# B&R Automation Studio project Parker_BMM_ST_V5_3147_V12 (part 19)

#### scrshot.c
```c
/********************************************************************
 * COPYRIGHT --  B&R China
 ********************************************************************
 * Program: length
 * File: length.c
 * Author: lijianjun
 * Created: March 06, 2013
 ********************************************************************
 * Implementation of program length --- parison length control
 ********************************************************************/

#include <bur/plctypes.h>

#ifdef _DEFAULT_INCLUDES
	#include <AsDefault.h>
#endif

#include <string.h>

/* Description: 	screen shot	(C language)	Library - VCScrsht										           */
/*------------------------------------------------------------------------------------------------------*/
/*				这个任务必须在循环7任务里，而且循环7的循环周期必须是1000ms，冗余时间为1000ms			       */
/*				It must also be inserted into Task Class #7 [1000 ms] and have a tolerance of 1000 ms.      */
/*  			程序员需要在初始化任务里定义device名称及相关信息就好了									           */
/*------------------------------------------------------------------------------------------------------*/
/*	version		author			date			decription
*********************************************************************************************************/

/********************************************************************************************************/
/*	<|> Variable to control this task:																                    */
/*		Name							Typ					Description									                    */
/*		step							| UINT				| screen shot step							                 //
//		DateTimeString_0			| DateTimeString	| output current date and time as string	              //
//		more see variable declaration																	                    */
/********************************************************************************************************/

/********************************************************************************************************/
/*	State commentary:																					      //
//			INIT:					   init step															   //
//			WAIT_USB_INSERT:		wait usb device insert												//
//			WAIT_COMMAND:    		wait for command													   //
//			INIT_SCREEN_SHOT:		Init screen shot													   //
//			SCREEN_SHOT:			Screen shot															   //
//			DEINIT_SCREEN_SHOT:		DeInit																//
//			ERROR_STEP:				Error step															   */

/********************************************************************************************************/
/*  Others:
//		指定首选存储介质:																				         //
//          在CPU属性里My Device定义介质名称															    //

//		截屏产生的文件名格式，以当前日期时间为文件名的bmp文件，DateTimeString_0.Date_Mode:		//
//				1:		美国时间格式USA date format  -- DateMM-DD-YYYY_TimeHH-MM-SS					  //
//				2:		亚洲时间格式Asia date format -- DateYYYY-MM-DD_TimeHH-MM-SS					  //
//				others:	默认模式Default format       -- DateDD-MM-YYYY_TimeHH-MM-SS				 //

//		建议：用fileio库来判断所在介质中是否有相同名称的文件，防止被覆盖								//
//		suggest: use filio to judge whether have a same name files in current diretory		  //

//		截屏状态gScreenShot.Status																		       //
//			0		等待存储介质插入插槽
			1		等待截屏开始指令
			2		截屏中
			3		截屏出错																			             //

*********************************************************************************************************/

/**********************************************************************************
**                          函数声明											 **
**********************************************************************************/

/**********************************************************************************
**                          宏定义												 **
**********************************************************************************/
#define INIT				         		0
#define WAIT_USB_INSERT		      		10
#define WAIT_DIR_SCREEN_CREATE		   20
#define WAIT_DIR_SINGLE_CREATE			40
#define WAIT_DIR_ALL_CREATE	   		50

#define WAIT_COMMAND		         100
#define INIT_SCREEN_SHOT	      110
#define SCREEN_SHOT			      120
#define DEINIT_SCREEN_SHOT	      140
#define ERROR_STEP			      200

/**********************************************************************************
**     	        		任务初始化								 				 **
**********************************************************************************/

_INIT  	void init()
{
	/*--------- 程序员根据实际，需要修改的代码 开始 ---------*/

	strcpy(gUSB_1.DeviceName, "USB_1");		/* 指定首选存储介质 */
	strcpy(gUSB_2.DeviceName, "USB_2");		/* 指定第二个选择存储介质 */

   strcpy(gUSB_1.DirScreenDeviceName, "SCREEN_1");		/* 指定首选存储介质目录 */
   strcpy(gUSB_2.DirScreenDeviceName, "SCREEN_2");		/* 指定第二个选择存储介质目录 */

   strcpy(dirScreenName,"ScreenShot");
   strcpy(dirSingleName,"SingleRecipe");
   strcpy(dirAllName,"AllRecipe");

   strcpy(gUSB_1.DirSingleDeviceName, "SINGLE_1");		/* 指定首选存储介质目录 */
   strcpy(gUSB_2.DirSingleDeviceName, "SINGLE_2");		/* 指定第二个选择存储介质目录 */

   strcpy(gUSB_1.DirAllDeviceName, "ALL_1");		/* 指定首选存储介质目录 */
   strcpy(gUSB_2.DirAllDeviceName, "ALL_2");		/* 指定第二个选择存储介质目录 */

	DateTimeString_0.Date_Mode = 2;		 	/* 截屏产生的文件名格式，见上面的说明 */

	statusUSB1 = 0;
	statusUSB2 = 0;

	gUSB_1.reserve = 0;
	gUSB_2.reserve = 0;

	/*--------- 程序员根据实际，需要修改的代码 结束 ---------*/
}/* _INIT  	void init() */

/**********************************************************************************
**     	        		任务循环部分							 				 **
**********************************************************************************/
_CYCLIC void cyclic()
{
   STRING NumName[5];

	/* 接收截屏开始指令 在别的任务里定义，原因：这个任务周期太长，有时抓不到信号 */
	gScreenShot.CmdScreenShot = gScreenShot.CmdScreenShot;

	gScreenShot.Status = gScreenShot.Status;/* 对外接口，截屏状态 */

	/*judge have a usb device insert or not*/
	/* 判断存储介质是否插入插槽内 */
	DirInfo_1.enable= 1;
	DirInfo_1.pDevice= (UDINT)(&gUSB_1.DeviceName);	/* 首选存储介质 */
	DirInfo_1.pPath= 0;							/* For Root, pPath is 0 */

	DirInfo(&DirInfo_1);

	if(DirInfo_1.status != ERR_FUB_BUSY)
	{
		if(DirInfo_1.status == ERR_OK)
		{
			statusUSB1 = 1;
		}
		else
		{
			if(DirInfo_1.status == fiERR_SYSTEM && ERR_FUB_BUSY == FileIoGetSysError())
			{
				statusUSB1 = 1;
			}
			else
			{
				statusUSB1 = 0;  /*  no usb  */
				gUSB_1.DeviceOk = 0;
				gUSB_1.reserve = 0;
			}
		}
	}/* if(DirInfo_1.status != ERR_FUB_BUSY) */

	if(1 == statusUSB1 && 0 == statusUSB1_old)
	{
		gUSB_1.reserve = 1;
	}

	statusUSB1_old = statusUSB1;

	DirInfo_2.enable= 1;
	DirInfo_2.pDevice= (UDINT)(&gUSB_2.DeviceName);
	DirInfo_2.pPath= 0;

	DirInfo(&DirInfo_2);

	if(DirInfo_2.status != ERR_FUB_BUSY)
	{
		if(DirInfo_2.status == ERR_OK)
		{
			statusUSB2 = 1;
		}
		else
		{
			if(DirInfo_2.status == fiERR_SYSTEM && ERR_FUB_BUSY == FileIoGetSysError())
			{
				statusUSB2 = 1;
			}
			else
			{
				statusUSB2 = 0;   /*  no usb  */
				gUSB_2.DeviceOk = 0;
				gUSB_2.reserve = 0;
			}
		}
	}/* if(DirInfo_2.status != ERR_FUB_BUSY) */

	if(1 == statusUSB2 && 0 == statusUSB2_old)
	{
		gUSB_2.reserve = 1;
	}

   if(0 == gUSB_2.DeviceOk && 0 == gUSB_1.DeviceOk)
   {
      if(1 == gScreenShot.CmdScreenShot)
      {
         gImply.NoUSB = 1;
         gScreenShot.CmdScreenShot = 0;
      }
   }
	/* 不在等待截屏指令状态， 如果谁发了截屏指令，无效 */
	if(gScreenShot.Status != 1)
	{
		gScreenShot.CmdScreenShot = 0;
		HideButton =1; //ipis1226
	}
	else
	{
		HideButton =0;	//ipis1226
	}

	/* 所有设备都没有准备好，就停在等待存储介质插入步 */
	if((gUSB_1.reserve == 0) && (gUSB_2.reserve == 0))
	{
		step = WAIT_USB_INSERT;
	}

	switch(step)
	{
		case INIT:				/* Init */
			gScreenShot.Status = 0;	/* 等待存储介质插入插槽 */
			step = WAIT_USB_INSERT;
			break;

		case WAIT_USB_INSERT:	/* wait for usb device insert */
			gScreenShot.Status = 0;	/* 等待存储介质插入插槽 */

			step = step;

			if((gUSB_1.reserve == 1) || (gUSB_2.reserve == 1))
			{
				step = WAIT_DIR_SCREEN_CREATE;
			}
			break;

      case WAIT_DIR_SCREEN_CREATE:
         if(gUSB_1.reserve == 1)
         {
            strcpy(deviceName, gUSB_1.DeviceName);
         }
         else if(gUSB_2.reserve == 1)
         {
            strcpy(deviceName, gUSB_2.DeviceName);
         }
         DirCreate_1.enable = 1;
         DirCreate_1.pDevice= (UDINT)(&deviceName);
         DirCreate_1.pName  = (UDINT)(&dirScreenName);

         /* Call FBK */
         DirCreate(&DirCreate_1);

         if(ERR_OK == DirCreate_1.status || fiERR_DIR_ALREADY_EXIST == DirCreate_1.status)
         {
            DirCreate_1.enable = 0;
            step = WAIT_DIR_SINGLE_CREATE;
         }
         else if(DirCreate_1.status != ERR_FUB_BUSY)
         {
				if(0 == strcmp(deviceName, gUSB_1.DeviceName))gUSB_1.reserve = 0;
				if(0 == strcmp(deviceName, gUSB_2.DeviceName))gUSB_2.reserve = 0;

            DirCreate_1.enable = 0;
            step = INIT;
         }
         break;

      case WAIT_DIR_SINGLE_CREATE:
         if(gUSB_1.reserve == 1)
         {
            strcpy(deviceName, gUSB_1.DeviceName);
         }
         else if(gUSB_2.reserve == 1)
         {
            strcpy(deviceName, gUSB_2.DeviceName);
         }
         DirCreate_1.enable = 1;
         DirCreate_1.pDevice= (UDINT)(&deviceName);
         DirCreate_1.pName  = (UDINT)(&dirSingleName);

         /* Call FBK */
         DirCreate(&DirCreate_1);

         if(ERR_OK == DirCreate_1.status || fiERR_DIR_ALREADY_EXIST == DirCreate_1.status)
         {
            DirCreate_1.enable = 0;
            step = WAIT_DIR_ALL_CREATE;
         }
         else if(DirCreate_1.status != ERR_FUB_BUSY)
         {
				if(0 == strcmp(deviceName, gUSB_1.DeviceName))gUSB_1.reserve = 0;
				if(0 == strcmp(deviceName, gUSB_2.DeviceName))gUSB_2.reserve = 0;

            DirCreate_1.enable = 0;
            step = INIT;
         }
         break;

      case WAIT_DIR_ALL_CREATE:
         if(gUSB_1.reserve == 1)
         {
            strcpy(deviceName, gUSB_1.DeviceName);
         }
         else if(gUSB_2.reserve == 1)
         {
            strcpy(deviceName, gUSB_2.DeviceName);
         }
         DirCreate_1.enable = 1;
         DirCreate_1.pDevice= (UDINT)(&deviceName);
         DirCreate_1.pName  = (UDINT)(&dirAllName);

         /* Call FBK */
         DirCreate(&DirCreate_1);

         if(ERR_OK == DirCreate_1.status || fiERR_DIR_ALREADY_EXIST == DirCreate_1.status)
         {
				if(0 == strcmp(deviceName, gUSB_1.DeviceName))gUSB_1.DeviceOk = 1;
				if(0 == strcmp(deviceName, gUSB_2.DeviceName))gUSB_2.DeviceOk = 1;

            DirCreate_1.enable = 0;
            step = WAIT_COMMAND;
         }
         else if(DirCreate_1.status != ERR_FUB_BUSY)
         {
				if(0 == strcmp(deviceName, gUSB_1.DeviceName))gUSB_1.reserve = 0;
				if(0 == strcmp(deviceName, gUSB_2.DeviceName))gUSB_2.reserve = 0;

            DirCreate_1.enable = 0;
            step = INIT;
         }
         break;

		case WAIT_COMMAND:		/* Wait for command */

			gScreenShot.Status = 1;	/* 等待截屏开始指令 */

			/* 允许客户按截屏开始按键 */
			gScreenShot.ScreenShotBtnStatus = gScreenShot.ScreenShotBtnStatus & (65535-2);

			if(gScreenShot.CmdScreenShot == 1)
			{
				gScreenShot.CmdScreenShot = 0;

				gScreenShot.ScreenShotBtnStatus = gScreenShot.ScreenShotBtnStatus | 2;

				/* Name format of Screen file: Year-month-day-hour-minute-second.bmp */
				DateTimeString_0.enable = 1;
				/*DateTimeString_0.Date_Mode = 2;		 Asia mode: DateYYYY-MM-DD_TimeHH-MM-SS */

            itoa((long)(gPanelObj.GetPicture),(unsigned long)NumName);

            strcpy(scrshotFileName,"Page_");

            strcat(scrshotFileName,NumName);

            strcat(scrshotFileName, "_");

            DateTimeString(&DateTimeString_0);

            strcat(scrshotFileName, DateTimeString_0.DisplayString);

            strcat(scrshotFileName, ".bmp");

				if(gUSB_1.DeviceOk == 1)
				{
					strcpy(deviceName, gUSB_1.DirScreenDeviceName);
				}
				else if(gUSB_2.DeviceOk == 1)
				{
					strcpy(deviceName, gUSB_2.DirScreenDeviceName);
				}
				step = INIT_SCREEN_SHOT;
			}
			break;

		case INIT_SCREEN_SHOT:	/* Init screen shot */

			gScreenShot.Status = 2;	/* 截屏中 */

			status = InitScreenShot(1, (UDINT)(&pHandle), (UDINT)(&scrshotFileName), (UDINT)(&deviceName), (UDINT)(&gPanelObj.VisualName));
			if(status == 0)
			{
				step = SCREEN_SHOT;
			}
			else
			{
				gScreenShot.errorNumber = status;
				step = ERROR_STEP;
			}
			break;

		case SCREEN_SHOT:		/* Screen shot */

			status = ScreenShot(1, pHandle);

			if(status != 1001)
			{
				if(status == 0)
				{
					step = DEINIT_SCREEN_SHOT;
				}
				else
				{
					gScreenShot.errorNumber = status;
					step = ERROR_STEP;
				}
			}
			break;

		case DEINIT_SCREEN_SHOT:/* DeInit screen shot */

			status = DeInitScreenShot(1, pHandle);

			if(status == 0)
			{
				step = WAIT_COMMAND;
			}
			else
			{
				gScreenShot.errorNumber = status;
				step = ERROR_STEP;
			}
			break;

		case ERROR_STEP:		/* Error step */

			gScreenShot.Status = 3;	/* 截屏出错 */
			step = INIT;
			break;
	}/* switch(step) */
}/* _CYCLIC void cyclic() */
```

#### scrshot.var
```iecst
VAR
	step : UINT;
	statusUSB1 : USINT;
	statusUSB1_old : USINT;
	statusUSB2 : USINT;
	statusUSB2_old : USINT;
	scrshotFileName : STRING[59];
	deviceName : STRING[19];
	DateTimeString_0 : DateTimeString;
	pHandle : UDINT;
	DirInfo_1 : DirInfo;
	DirInfo_2 : DirInfo;
	DirCreate_1 : DirCreate;
	dirScreenName : STRING[19];
	dirSingleName : STRING[19];
	dirAllName : STRING[19];
	status : UINT;
	HideButton : USINT; (*ipis1226*)
END_VAR
```

### Program Logical/screen/password (ANSIC, version 1.00.0) - password login modify

#### password.c
```c
/********************************************************************
 * COPYRIGHT --  B&R China
 ********************************************************************
 * Program: password
 * File: password.c
 * Author: lijianjun
 * Created: March 06, 2013
 ********************************************************************
 * Implementation of program password --- password control
 ********************************************************************/

#include <bur/plctypes.h>
#include <string.h>

#ifdef _DEFAULT_INCLUDES
	#include <AsDefault.h>
#endif

#include "pic_id.h"

/**************************************************************************************
** 					 	 dedine								              			 **
**************************************************************************************/
#define S$STEP_INIT_OK     10000

#define S$STEP_IDLE        100
#define S$STEP_READ        1000
#define S$STEP_WRITE       2000

#define S$STEP_ERROR	      30000

/**************************************************************************************
** 							         function declare  				  			             **
**************************************************************************************/
void Pwd_Set(unsigned short picGet,unsigned short  picObj);
/**************************************************************************************
*     	        		      I N I T U P  O F   T H E   T A S K 		 				       **
**************************************************************************************/

_INIT  void Pwd_init( void )
{
	InputCompletion = 0;

	strcpy(gPwd.PwdInput,   "           ");    	/*  11 space char  */
	strcpy(gPwd.HisPwdInput,"           ");		/*  11 space char  */

	DataObjOperate.InitStep = 100;
}
/**************************************************************************************
*        				    C Y C L I C   P A R T   O F   T H E   T A S K  				  *
**************************************************************************************/

_CYCLIC  void Pwd_cyclic ( void )
{

	if (gPasswordLogout)  //ipis0218
	{
		InputCompletion =1;
		strcpy(gPwd.PwdInput,   "           ");    	/*  11 space char  */
		gPasswordLogout =0;
	}

	gPanelObj.PasswordLevel = gPwd.PwdLevel;

	switch(DataObjOperate.InitStep)
	{
		case 100:
			DataObjOperate.Ident = 0;

			DatObj_Info.enable = 1;
			DatObj_Info.pName  =(unsigned long)("pwddata");
			DatObjInfo(&DatObj_Info);

			if(doERR_MODULNOTFOUND == DatObj_Info.status)
			{
				DataObjOperate.InitStep = 200;
			}
			else if(0 == DatObj_Info.status)
			{
				DataObjOperate.Ident    = DatObj_Info.ident;
				DataObjOperate.InitStep = 800;
			}
			else
			{
				DataObjOperate.InitStep = S$STEP_ERROR;
			}
			break;
		case 200:                              	/* create data module */
			DatObj_Create.enable   = 1;
			DatObj_Create.pName    = DatObj_Info.pName;
			DatObj_Create.len      = sizeof(Pwd_typ);
			DatObj_Create.MemType  = doUSRROM;
			DatObj_Create.Option   = 0;
			DatObj_Create.pCpyData = 0;

			DataObjOperate.InitStep = 300;
			break;
		case 300:
			DatObjCreate(&DatObj_Create);
			if(0 == DatObj_Create.status)
			{
				DataObjOperate.Ident = DatObj_Create.ident;
				DataObjOperate.InitStep = 400;
			}
			break;
		case 400:
			memset(&gPwd,0,sizeof(Pwd_typ));

			strcpy(gPwd.Level[2],"8888");
			strcpy(gPwd.Level[1],"7777");
			strcpy(gPwd.Level[0],"6666");

			gPwd.length_1 = 120;
			gPwd.length_2 = 120;
			gPwd.length_3 = 120;

			strcpy(gPwd.Pwd_1,"0098768876");
			strcpy(gPwd.Pwd_2,"0098768872");
			strcpy(gPwd.Pwd_3,"0098768870");

			strcpy(gPwd.PwdInput,   "           ");    	 	 /*  11 space char  */
			strcpy(gPwd.HisPwdInput,"           ");			/*  11 space char  */

			DataObjOperate.InitStep = 500;
			break;
		case 500:
			DatObj_Write.enable  = 1;
			DatObj_Write.ident	 = DataObjOperate.Ident;
			DatObj_Write.pSource = (unsigned long )&gPwd;
			DatObj_Write.len     = sizeof(Pwd_typ);

			DataObjOperate.InitStep = 600;
			break;
		case 600:
			DatObjWrite(&DatObj_Write);
			if(0 == DatObj_Write.status)
			{
				DataObjOperate.InitStep = 700;
			}
			else
			{
				DataObjOperate.InitStep = S$STEP_ERROR;
			}
			break;
		case 700:
			DataObjOperate.InitStep = 1000;
			break;
		case 800:
			DatObj_Read.enable 		 = 1;
			DatObj_Read.ident 		 = DataObjOperate.Ident ;
			DatObj_Read.Offset 		 = 0;
			DatObj_Read.pDestination = (unsigned long )&gPwd;
			DatObj_Read.len 		 = sizeof(Pwd_typ);

			DataObjOperate.InitStep = 900;
			break;
		case 900:
			DatObjRead(&DatObj_Read);
			if(0 == DatObj_Read.status)
			{
				DataObjOperate.InitStep = 1000;
			}
			else
			{
				DataObjOperate.InitStep = S$STEP_ERROR;
			}
			break;
		case 1000:
			gPwd.PwdLevel = 0;

			strcpy(gPwd.PwdInput,   "           ");    	/*  11 space char  */
			strcpy(gPwd.HisPwdInput,"           ");	    /*  11 space char  */

			DataObjOperate.Step = S$STEP_IDLE;
			DataObjOperate.InitStep = S$STEP_INIT_OK;
			break;
		case S$STEP_ERROR:
			break;
		default:
			break;
	}/* switch(DataObjOperate.InitStep) */

	if(DataObjOperate.Ident != 0 && DataObjOperate.InitStep == S$STEP_INIT_OK )
	{
		switch(DataObjOperate.Step )
		{
			case S$STEP_IDLE:
				if(1 == gPwd.wSavePassword)
				{
					gPwd.wSavePassword = 0;
					DataObjOperate.Step = S$STEP_WRITE;
				}
				break;
			case S$STEP_WRITE:
				DatObj_Write.enable  = 1;
				DatObj_Write.ident	 = DataObjOperate.Ident;
				DatObj_Write.pSource = (unsigned long )&gPwd;
				DatObj_Write.len     = sizeof(Pwd_typ);

				DataObjOperate.Step = S$STEP_WRITE + 100;
				break;
			case (S$STEP_WRITE + 100):
				DatObjWrite(&DatObj_Write);
				if(0 == DatObj_Write.status)
				{
					DataObjOperate.Step = S$STEP_WRITE + 200;
				}
				break;
			case (S$STEP_WRITE + 200):
				DataObjOperate.Step = S$STEP_IDLE;
				break;
			default:
				break;
		}/* switch(DataObjOperate.Step) */

		WorkingDays = 0;

		if(1 == gPwd.Option[0] && 0 == gPwd.OK_1)
		{
			WorkingDays = WorkingDays + gPwd.length_1;
		}
		else if(1 == gPwd.Option[1] && 0 == gPwd.OK_2)
		{
			WorkingDays = WorkingDays + gPwd.length_2;
		}
		else if(1 == gPwd.Option[2] && 0 == gPwd.OK_3)
		{
			WorkingDays = WorkingDays + gPwd.length_3;
		}

		if(0 == WorkingDays)
		{
			gMachineInfo.TimeStopMachine = 0;
		}
		else
		{
			if(gMachineStopDays > WorkingDays)
			{
				gMachineInfo.TimeStopMachine = 1;
			}
			else
			{
				gMachineInfo.TimeStopMachine = 0;
			}
		}

		if(gAlarm.batteryLow)
		{
			gMachineInfo.TimeStopMachine = 0;
		}

		if(PIC_PASSWORD_LOGIN == gPanelObj.GetPicture || PIC_INIT == gPanelObj.GetPicture)
		{
			if(1 == InputCompletion)
			{
				InputCompletion = 0;
				strcpy(gPwd.HisPwdInput,gPwd.PwdInput);
				strcpy(gPwd.PwdInput,"           ");		/*  11 space char  */

				if( !strcmp(gPwd.HisPwdInput,gPanelObj.PasswordHigh))
				{
			   		gPwd.PwdLevel = 5;
			   	}
				else if( !strcmp(gPwd.HisPwdInput,gPanelObj.Password4))
				{
			   		gPwd.PwdLevel = 4;
			   	}
				else if(!strcmp(gPwd.HisPwdInput,gPwd.Level[2]))
				{
					gPwd.PwdLevel = 3;
				//	gPwd.PwdLevel = 4;  //ipis0226
				}
				else if(!strcmp(gPwd.HisPwdInput,gPwd.Level[1]))
				{
					gPwd.PwdLevel = 2;
				}
				else if(!strcmp(gPwd.HisPwdInput,gPwd.Level[0]))
				{
					gPwd.PwdLevel = 1;
				}
				else
				{
					if(PIC_PASSWORD_LOGIN == gPanelObj.GetPicture)
					{
						if(!strcmp(gPwd.HisPwdInput,gPwd.Pwd_3))
						{
							if(1 == gPwd.Option[2])
							{
								gMachineStopDays = 0;
								gPwd.OK_3 = 1;
								gPwd.OK_2 = 1;
								gPwd.OK_1 = 1;
								gPwd.wSavePassword = 1;
							}
						}
						else if (!strcmp(gPwd.HisPwdInput,gPwd.Pwd_2))
						{
							if(1 == gPwd.Option[1])
							{
								gMachineStopDays = 0;
								gPwd.OK_2 = 1;
								gPwd.OK_1 = 1;
								gPwd.wSavePassword = 1;
							}
						}
						else if (!strcmp(gPwd.HisPwdInput,gPwd.Pwd_1))
						{
							if(1 == gPwd.Option[0])
							{
								gMachineStopDays = 0;
								gPwd.OK_1 = 1;
								gPwd.wSavePassword = 1;
							}
						}
					}/* if(PIC_PASSWORD_LOGIN == gPanelObj.GetPicture) */
					gPwd.PwdLevel = 0;
				}
			}/* if(1 == InputCompletion */
		}/* if(gPanelObj.GetPicture == PIC_PASSWORD_LOGIN || PIC_INIT_PIC == gPanelObj.GetPicture ) */

		Pwd_Set(gPanelObj.GetPicture,PIC_PASSWORD_SET);

	}/* if(DataObjOperate.Ident != 0 && DataObjOperate.InitStep == S$STEP_INIT_OK ) */
}
/**************************************************************************************
** 							Function Realization  				  			         **
**************************************************************************************/

void Pwd_Set(UINT picGet,UINT picObj)
{
	short	i;

 	if (picGet != picObj)
 	{
		gPwd.StatusOfPasswordSet = 0;
		for (i=0;i<=2;i++)
		{
			strcpy(gPwd.PasswordSet[i],   "           ");
			strcpy(gPwd.HisPasswordSet[i],"           ");
		}
 		return;
 	}

 	for (i=0;i<=2;i++)
 	{

 		if(1 == gPwd.CompletionHisPasswordSet[i])
 		{
 			gPwd.StatusOfPasswordSet         = 1;
 			gPwd.CompletionHisPasswordSet[i] = 0;
 		}

 		if(1 == gPwd.CompletionPasswordSet[i])
	 	{
	 		if (strcmp(gPwd.PasswordSet[i] ,"           ")!= 0)
		    {
			    if (0 == strcmp(gPwd.PasswordSet[i],gPwd.HisPasswordSet[i]))
				{
					gPwd.StatusOfPasswordSet  = 2; /* setting ok */
		    		gPwd.wSavePassword	  	 = 1;
		    		strcpy(gPwd.Level[i],gPwd.PasswordSet[i]);

					strcpy(gPwd.PasswordSet[i],   "           ");
					strcpy(gPwd.HisPasswordSet[i],"           ");

		    	}
	    		else
	    		{
	    			gPwd.StatusOfPasswordSet = 3; /* setting failed */

	 				strcpy(gPwd.PasswordSet[i],   "           ");
					strcpy(gPwd.HisPasswordSet[i],"           ");
	    		}
	    	}
			gPwd.CompletionPasswordSet[i] = 0;
	 	}/* if(1 == gPwd.CompletionPasswordSet[i]) */
	}/* for (i=0;i<=2;i++) */
 }/* end of function */
```

#### password.var
```iecst
VAR
	DatObj_Info	:DatObjInfo;
	DatObj_Create	:DatObjCreate;
	DatObj_Write	:DatObjWrite;
	DatObj_Read	:DatObjRead;
	DataObjOperate	:DatObj_Operate_typ;
    InputCompletion	:USINT;

    WorkingDays : UDINT;
END_VAR
```

### Program Logical/screen/vpn (ANSIC, version 1.00.0) - IP configure

#### vpn.c
```c
/********************************************************************
 * COPYRIGHT --  B&R China
 ********************************************************************
 * Program: vpn
 * File: vpn.c
 * Author: lijianjun
 * Created: March 06, 2013
 ********************************************************************
 * Implementation of program vpn --- ip address control
 ********************************************************************/

#include <bur/plctypes.h>

#ifdef _DEFAULT_INCLUDES
#include <AsDefault.h>
#endif

#include <string.h>

//#include "keyap880.h"
#include "keyap2100.h"
#include "pic_id.h"

char substring(char *dst,char *src,int start,int len);

/********************************************************************************************************/
/*  Others:
	vpn.FlagManualSetIP：0=自动获取IP地址类型，1=手动设置IP地址
	vpn存放当前IP地址，子网掩码，网关地址等，以及手动设置IP地址，子网掩码，网关地址等参数，

		typedef struct
		{
			BOOL			FlagManualSetIP;		* 标志位：1 = 手动设定IP地址 *
			BOOL			CmdSetIP;				* 设置IP地址指令 *
			BOOL			CmdSetSubnetMark;		* 设置子网掩码指令 *
			BOOL			CmdSetGateway;			* 设置网关地址指令 *

			STRING			CurrentIPString[16];	* 当前IP地址 *
			STRING			CurrentSubnetMarkString[16];* 当前子网掩码 *
			STRING			CurrentGatewayString[16];* 当前网关地址 *

			Address_typ		ParaSetIP;				* 手动设置IP地址模式下，IP地址参数 *
			Address_typ		ParaSetSubnetMark;		* 手动设置IP地址模式下，子网掩码参数 *
			Address_typ		ParaSetGateway;			* 手动设置IP地址模式下，网关地址参数 *

		}VPN_typ;

*********************************************************************************************************/

/**********************************************************************************
**                          宏定义												 **
**********************************************************************************/
#define INIT				       0
#define GET_ETH_CFG_MODE	   10
#define GET_ETH_CFG_ADR	      20
#define GET_ETH_CFG_SUBNET	   30
#define GET_ETH_CFG_GATEWAY 	40

#define WAIT_COMMAND          100
#define SET_ETH_CFG_MODE		110
#define SET_ETH_CFG_ADR	      120
#define SET_ETH_CFG_SUBNET 	130
#define SET_ETH_CFG_GATEWAY   140
#define ERROR_STEP            9999

/**********************************************************************************
**     	        		I N I T U P  O F   T H E   T A S K 		 				 **
**********************************************************************************/
_INIT void init()
{
	/*------------- 编程人员根据实际需要修改的地方 开始 -----------------*/

	strcpy(vpnDevice,"IF3");	/*指定VPN使用的端口*/

	/*------------- 编程人员根据实际需要修改的地方 结束 -----------------*/
	step = INIT;

	bGetCurrentIP_USINT = 1;

}/* _INIT void init() */

/**********************************************************************************
**        			C Y C L I C   P A R T   O F   T H E   T A S K  				 **
**********************************************************************************/
_CYCLIC void cyclic()
{
	if(gPanelObj.GetPicture == PIC_IP_CONFIG && step == WAIT_COMMAND)
	{
		F5_bHiden = 0;
	}
	else
	{
		F5_bHiden = 1;
	}

	/*-------------- 判断手自动模式是否切换了 -------------------------*/
	R_TRIG_KeyF5.CLK = gPanelObj.KeyMatric[S$KEYMATRIX_F5];
		R_TRIG(&R_TRIG_KeyF5);

	/*if(1 == R_TRIG_KeyF5.Q)
	{
		if(gPanelObj.GetPicture == PIC_IP_CONFIG)
		{
			if(0 == F5_bHiden)
			{
				if( cfgCONFIGMODE_MANUALLY == vpn.CurrentConfigMode)
				{
					vpn.ParaSetConfigMode = cfgCONFIGMODE_DHCPCLIENT;
				}
				else
				{
					vpn.ParaSetConfigMode = cfgCONFIGMODE_MANUALLY;
				}
				vpn.CmdSetMode = 1;
			}
		}
	}*//* if(1 == R_TRIG_KeyF5.Q) */

	vpn.ParaSetConfigMode = cfgCONFIGMODE_MANUALLY;

	switch(step)
	{
		case INIT:				/*初始化*/
			step = GET_ETH_CFG_MODE;
			break;

		case GET_ETH_CFG_MODE:	/*读当前配置模式*/
			CfgGetEthConfigMode_0.pDevice = (UDINT)&vpnDevice[0];
			CfgGetEthConfigMode_0.enable  = 1;

			CfgGetEthConfigMode(&CfgGetEthConfigMode_0);

			if(ERR_FUB_BUSY != CfgGetEthConfigMode_0.status)
			{
				if(ERR_OK == CfgGetEthConfigMode_0.status)
				{
					if(cfgCONFIGMODE_MANUALLY == CfgGetEthConfigMode_0.ConfigMode)
					{
						vpn.FlagManualSetIP = 1;
						step = GET_ETH_CFG_ADR;
					}
					else if(cfgCONFIGMODE_DHCPCLIENT == CfgGetEthConfigMode_0.ConfigMode)
					{
						vpn.FlagManualSetIP = 0;
						step = GET_ETH_CFG_ADR;
					}
					vpn.CurrentConfigMode = CfgGetEthConfigMode_0.ConfigMode;
				}
				else
				{
					step = ERROR_STEP;
				}
			}
			break;

		case GET_ETH_CFG_ADR:		/*读当前IP地址*/
			CfgGetIPAddr_0.pDevice = (UDINT)&vpnDevice[0];
			CfgGetIPAddr_0.pIPAddr = (UDINT)&vpn.CurrentIPString[0];
			CfgGetIPAddr_0.Len     = 16;
			CfgGetIPAddr_0.enable  = 1;

			CfgGetIPAddr(&CfgGetIPAddr_0);

			if(ERR_FUB_BUSY != CfgGetIPAddr_0.status)
			{
				if(ERR_OK == CfgGetIPAddr_0.status)
				{
					step = GET_ETH_CFG_SUBNET;
				}
				else
				{
					step = ERROR_STEP;
				}
			}
			break;

		case GET_ETH_CFG_SUBNET:		/*读当前子网掩码*/
			CfgGetSubnetMask_0.pDevice = (UDINT)&vpnDevice[0];
			CfgGetSubnetMask_0.pSubnetMask = (UDINT)&vpn.CurrentSubnetMarkString[0];
			CfgGetSubnetMask_0.Len     = 16;
			CfgGetSubnetMask_0.enable  = 1;

			CfgGetSubnetMask(&CfgGetSubnetMask_0);

			if(ERR_FUB_BUSY != CfgGetSubnetMask_0.status)
			{
				if(ERR_OK == CfgGetSubnetMask_0.status)
				{
					step = GET_ETH_CFG_GATEWAY;
				}
				else
				{
					step = ERROR_STEP;
				}
			}
			break;

		case GET_ETH_CFG_GATEWAY:		/*读当前默认网关*/
			CfgGetDefaultGateway_0.pDevice = (UDINT)&vpnDevice[0];
			CfgGetDefaultGateway_0.pGateway= (UDINT)&vpn.CurrentGatewayString[0];
			CfgGetDefaultGateway_0.Len     = 16;
			CfgGetDefaultGateway_0.enable  = 1;

			CfgGetDefaultGateway(&CfgGetDefaultGateway_0);

			if(ERR_FUB_BUSY != CfgGetDefaultGateway_0.status)
			{
				if(ERR_OK == CfgGetDefaultGateway_0.status)
				{
					step = WAIT_COMMAND;
				}
				else
				{
					if(cfgERR_PARAM_NOT_SET == CfgGetDefaultGateway_0.status)
					{
						step = WAIT_COMMAND;
					}
					else
					{
						step = ERROR_STEP;
					}
				}
			}
			break;

		case WAIT_COMMAND:
			if(0 == vpn.FlagManualSetIP)
			{
				vpn.CmdSetIP         = 0;
				vpn.CmdSetSubnetMark = 0;
				vpn.CmdSetGateway    = 0;

				if(1 == vpn.CmdSetMode)
				{
					vpn.CmdSetMode = 0;
					step = SET_ETH_CFG_MODE;
				}
				else
				{
					step = GET_ETH_CFG_MODE;
				}
			}
			else
			{
				if(1 == vpn.CmdSetMode)
				{
					vpn.CmdSetMode = 0;
					step = SET_ETH_CFG_MODE;
				}
				else
				{
					if(1 == vpn.CmdSetIP)
					{
						vpn.CmdSetIP = 0;
						step = SET_ETH_CFG_ADR;
					}
					else if(1 == vpn.CmdSetSubnetMark)
					{
						vpn.CmdSetSubnetMark = 0;
						step = SET_ETH_CFG_SUBNET;
					}
					else if(1 == vpn.CmdSetGateway)
					{
						vpn.CmdSetGateway = 0;
						step = SET_ETH_CFG_GATEWAY;
					}
				}/* if(1 == vpn.CmdSetMode) */
			}/* if(0 == vpn.FlagManualSetIP) */
			break;

		case SET_ETH_CFG_MODE:		/*设定配置模式*/
			CfgSetEthConfigMode_0.pDevice = (UDINT)&vpnDevice[0];

			CfgSetEthConfigMode_0.ConfigMode = vpn.ParaSetConfigMode;
			CfgSetEthConfigMode_0.Option  = cfgOPTION_VOLATILE;

			CfgSetEthConfigMode_0.enable  = 1;

			CfgSetEthConfigMode(&CfgSetEthConfigMode_0);

			if(ERR_FUB_BUSY != CfgSetEthConfigMode_0.status)
			{
				if(ERR_OK == CfgSetEthConfigMode_0.status)
				{
					step = GET_ETH_CFG_MODE;
				}
				else
				{
					step = ERROR_STEP;
				}
			}
			break;

		case SET_ETH_CFG_ADR:		/*设定IP*/
			itoa(vpn.ParaSetIP.Address3, (UDINT)&tempString);
			strcpy(setIPString, tempString);

			strcat(setIPString, ".");

			itoa(vpn.ParaSetIP.Address2, (UDINT)&tempString);
			strcat(setIPString, tempString);

			strcat(setIPString, ".");

			itoa(vpn.ParaSetIP.Address1, (UDINT)&tempString);
			strcat(setIPString, tempString);

			strcat(setIPString, ".");

			itoa(vpn.ParaSetIP.Address0, (UDINT)&tempString);
			strcat(setIPString, tempString);

			CfgSetIPAddr_0.pDevice = (UDINT)&vpnDevice[0];
			CfgSetIPAddr_0.pIPAddr = (UDINT)&setIPString[0];
			CfgSetIPAddr_0.Option  = cfgOPTION_NON_VOLATILE;
			CfgSetIPAddr_0.enable  = 1;

			CfgSetIPAddr(&CfgSetIPAddr_0);

			if(ERR_FUB_BUSY != CfgSetIPAddr_0.status)
			{
				if(ERR_OK == CfgSetIPAddr_0.status)
				{
					step = GET_ETH_CFG_MODE;

					/*update fix*/
					gUserFix.ProjectInfo.Address3 = vpn.ParaSetIP.Address3;
					gUserFix.ProjectInfo.Address2 = vpn.ParaSetIP.Address2;
					gUserFix.ProjectInfo.Address1 = vpn.ParaSetIP.Address1;
					gUserFix.ProjectInfo.Address0 = vpn.ParaSetIP.Address0;

					gRecipeOperate.OnceSave = 1;
				}
				else
				{
					step = ERROR_STEP;
				}
			}
			break;

		case SET_ETH_CFG_SUBNET:		/*设定子网掩码*/
			itoa(vpn.ParaSetSubnetMark.Address3, (UDINT)&tempString);
			strcpy(setSubnetMarkString, tempString);

			strcat(setSubnetMarkString, ".");

			itoa(vpn.ParaSetSubnetMark.Address2, (UDINT)&tempString);
			strcat(setSubnetMarkString, tempString);

			strcat(setSubnetMarkString, ".");

			itoa(vpn.ParaSetSubnetMark.Address1, (UDINT)&tempString);
			strcat(setSubnetMarkString, tempString);

			strcat(setSubnetMarkString, ".");

			itoa(vpn.ParaSetSubnetMark.Address0, (UDINT)&tempString);
			strcat(setSubnetMarkString, tempString);

			CfgSetSubnetMask_0.pDevice = (UDINT)&vpnDevice[0];
			CfgSetSubnetMask_0.pSubnetMask = (UDINT)&setSubnetMarkString[0];
			CfgSetSubnetMask_0.Option  = cfgOPTION_NON_VOLATILE;
			CfgSetSubnetMask_0.enable  = 1;

			CfgSetSubnetMask(&CfgSetSubnetMask_0);

			if(ERR_FUB_BUSY != CfgSetSubnetMask_0.status)
			{
				if(ERR_OK == CfgSetSubnetMask_0.status)
				{
					step = GET_ETH_CFG_MODE;
				}
				else
				{
					step = ERROR_STEP;
				}
			}
			break;

		case SET_ETH_CFG_GATEWAY:		/*设定网关*/
			itoa(vpn.ParaSetGateway.Address3, (UDINT)&tempString);
			strcpy(setGatewayString, tempString);

			strcat(setGatewayString, ".");

			itoa(vpn.ParaSetGateway.Address2, (UDINT)&tempString);
			strcat(setGatewayString, tempString);

			strcat(setGatewayString, ".");

			itoa(vpn.ParaSetGateway.Address1, (UDINT)&tempString);
			strcat(setGatewayString, tempString);

			strcat(setGatewayString, ".");

			itoa(vpn.ParaSetGateway.Address0, (UDINT)&tempString);
			strcat(setGatewayString, tempString);

			CfgSetDefaultGateway_0.pDevice = (UDINT)&vpnDevice[0];
			CfgSetDefaultGateway_0.pGateway = (UDINT)&setGatewayString[0];
			CfgSetDefaultGateway_0.Option  = cfgOPTION_NON_VOLATILE;
			CfgSetDefaultGateway_0.enable  = 1;

			CfgSetDefaultGateway(&CfgSetDefaultGateway_0);

			if(ERR_FUB_BUSY != CfgSetDefaultGateway_0.status)
			{
				if(ERR_OK == CfgSetDefaultGateway_0.status)
				{
					step = GET_ETH_CFG_MODE;
				}
				else
				{
					step = ERROR_STEP;
				}
			}
			break;

		case ERROR_STEP:	/*error step*/
			step = 0;
			break;

		default:
			break;
	}/* switch(step) */

	/*Get config ip*/
	if(bGetCurrentIP_USINT)
	{
		bGetCurrentIP_USINT = 0;
		Part_num_count = 0;
		Char_num = 0;
		old_Char_num = 0;
		for (ii = 0; ii < sizeof(vpn.CurrentIPString); ii++)
		{
			Charr = (char*)(vpn.CurrentIPString[ii]);

			if( Charr == 46)
			{
				Char_num = ii;

				switch (Part_num_count)
				{
					case 0:
						substring(sTempAddress3,vpn.CurrentIPString,0,Char_num);
						old_Char_num = Char_num;
						break;
					case 1:
						substring(sTempAddress2,vpn.CurrentIPString,old_Char_num+1,Char_num-old_Char_num-1);
						old_Char_num = Char_num;
						break;
					case 2:
						substring(sTempAddress1,vpn.CurrentIPString,old_Char_num+1,Char_num-old_Char_num-1);
						old_Char_num = Char_num;
						break;
				}
				Part_num_count++;
			}
			if(Part_num_count == 3)
			{
				substring(sTempAddress0,vpn.CurrentIPString,old_Char_num+1,sizeof(vpn.CurrentIPString)-old_Char_num);
			}

		}

		uConfigAddress3 = atoi((UDINT) &sTempAddress3);
		uConfigAddress2 = atoi((UDINT) &sTempAddress2);
		uConfigAddress1 = atoi((UDINT) &sTempAddress1);
		uConfigAddress0 = atoi((UDINT) &sTempAddress0);

		/*check current vs fix (if different than excute set ip cmd)*/
		if(gUserFix.ProjectInfo.Address0 != uConfigAddress0
			|| gUserFix.ProjectInfo.Address1 != uConfigAddress1
			|| gUserFix.ProjectInfo.Address2 != uConfigAddress2
			|| gUserFix.ProjectInfo.Address3 != uConfigAddress3
			)
		{
			vpn.ParaSetIP.Address0 = gUserFix.ProjectInfo.Address0;
			vpn.ParaSetIP.Address1 = gUserFix.ProjectInfo.Address1;
			vpn.ParaSetIP.Address2 = gUserFix.ProjectInfo.Address2;
			vpn.ParaSetIP.Address3 = gUserFix.ProjectInfo.Address3;

			vpn.CmdSetIP = 1;
		}
	}
}/* _CYCLIC void cyclic() */

char substring(char *dst,char *src,int start,int len)
{
	char *p=dst;
	char *q=src;
	int length=strlen(src);
	if(start>=length||start<0)
		return NULL;
	if(len>length)
		len=length-start;
	q+=start;
	while(len--)
	{
		*(p++)=*(q++);
	}
	*(p++)='\0';
	return dst;
}
```

#### vpn.var
```iecst
VAR
	vpn : VPN_typ;
	step : UINT;
	setIPString : STRING[15];
	setSubnetMarkString : STRING[15];
	setGatewayString : STRING[15];
	vpnDevice : STRING[15];
	tempString : STRING[3];
	CfgGetIPAddr_0 : CfgGetIPAddr;
	CfgGetSubnetMask_0 : CfgGetSubnetMask;
	CfgGetDefaultGateway_0 : CfgGetDefaultGateway;
	CfgGetEthConfigMode_0 : CfgGetEthConfigMode;
	CfgSetIPAddr_0 : CfgSetIPAddr;
	CfgSetSubnetMask_0 : CfgSetSubnetMask;
	CfgSetDefaultGateway_0 : CfgSetDefaultGateway;
	CfgSetEthConfigMode_0 : CfgSetEthConfigMode;
	R_TRIG_KeyF5 : R_TRIG;
	F5_bHiden : UINT;
END_VAR
(*Fix IP*)
VAR
	bGetCurrentIP_USINT : BOOL;
	Charr : BYTE;
	ii : USINT;
	sTempAddress1 : STRING[3];
	sTempAddress2 : STRING[3];
	sTempAddress3 : STRING[3];
	sTempAddress0 : STRING[3];
	Char_num : USINT;
	old_Char_num : USINT;
	Part_num_count : USINT;
	uConfigAddress0 : USINT;
	uConfigAddress1 : USINT;
	uConfigAddress2 : USINT;
	uConfigAddress3 : USINT;
END_VAR
```

#### vpn.typ - Local data types
```iecst
(********************************************************************
 * COPYRIGHT --  B&R
 ********************************************************************
 * Program: vpn
 * File: vpn.typ
 * Author: lij
 * Created: March 06, 2013
 ********************************************************************
 * Local data types of program vpn
 ********************************************************************)

TYPE
	Address_typ : 	STRUCT
		Address3 : USINT;
		Address2 : USINT;
		Address1 : USINT;
		Address0 : USINT;
END_STRUCT;
	VPN_typ : 	STRUCT
		FlagManualSetIP : BOOL;
		CmdSetMode : BOOL;
		CmdSetIP : BOOL;
		CmdSetSubnetMark : BOOL;
		CmdSetGateway : BOOL;
		Reserve2 : BOOL;
		Reserve1 : BOOL;
		Reserve0 : BOOL;
		CurrentConfigMode : UDINT;
		CurrentIPString : STRING[15];
		CurrentSubnetMarkString : STRING[15];
		CurrentGatewayString : STRING[15];
		ParaSetConfigMode : UDINT;
		ParaSetIP : Address_typ;
		ParaSetSubnetMark : Address_typ;
		ParaSetGateway : Address_typ;
END_STRUCT;
END_TYPE
```

### Program Logical/screen/panel (ANSIC, version 1.00.0) - panel display
